SUBAPPLICATION Uebung_036 (* Spiegelabfolge V2 mit Schrittkette *)
  (* Standard: 61499-2; Description: Copyright (c) 2023 Meisterschulen am Ostbahnhof This program and the accompanying materials are made available under the terms of the Eclipse Public License 2.0 which is available at https://www.eclipse.org/legal/epl-2.0/ SPDX-License-Identifier: EPL-2.0 *)
  (* Version 1.0, 2023-10-23, Franz Höpfinger, Meisterschulen am Ostbahnhof *)
  PACKAGE Uebungen;
  IMPORT Uebungen::const::UT::DefaultPool::OutputNumber_N1;
  IMPORT logiBUS::io::DI::logiBUS_DI::Input_I1;
  IMPORT logiBUS::io::DI::logiBUS_DI::Input_I2;
  IMPORT logiBUS::io::DI::logiBUS_DI::Input_I3;
  IMPORT logiBUS::io::DI::logiBUS_DI::Input_I4;
  IMPORT logiBUS::io::DI::logiBUS_DI_Events::BUTTON_SINGLE_CLICK;
  IMPORT logiBUS::io::DQ::logiBUS_DO::Output_Q1;
  IMPORT logiBUS::io::DQ::logiBUS_DO::Output_Q2;
  IMPORT logiBUS::io::DQ::logiBUS_DO::Output_Q3;
  IMPORT logiBUS::io::DQ::logiBUS_DO::Output_Q4;
  IMPORT logiBUS::utils::sequence::const::sequence::NO_TIME;
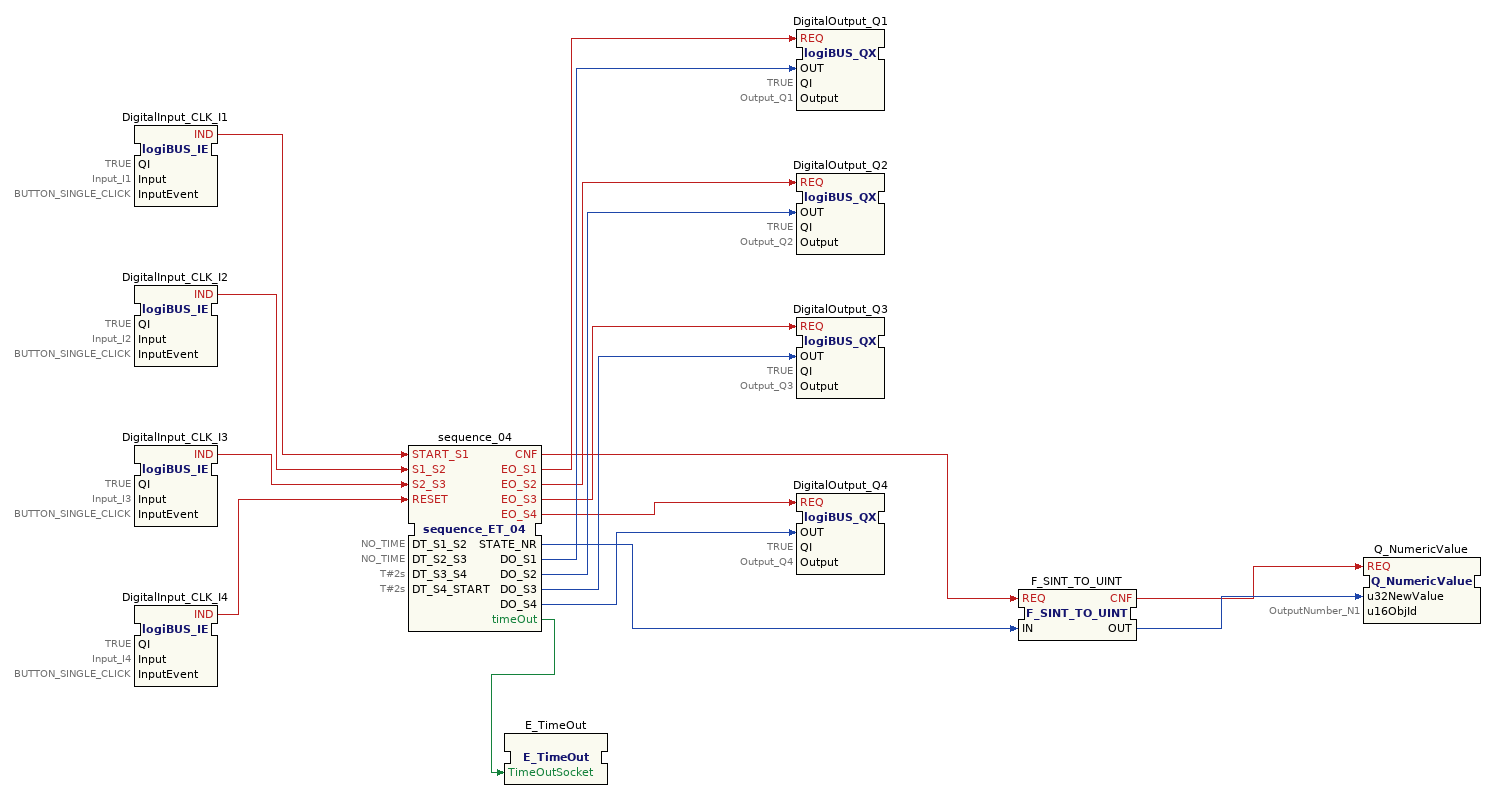
  FBS
    DigitalOutput_Q1 : logiBUS::io::DQ::logiBUS_QX(QI := TRUE, Output := Output_Q1);
    E_TimeOut : iec61499::events::E_TimeOut;
    DigitalOutput_Q2 : logiBUS::io::DQ::logiBUS_QX(QI := TRUE, Output := Output_Q2);
    DigitalOutput_Q3 : logiBUS::io::DQ::logiBUS_QX(QI := TRUE, Output := Output_Q3);
    DigitalOutput_Q4 : logiBUS::io::DQ::logiBUS_QX(QI := TRUE, Output := Output_Q4);
    DigitalInput_CLK_I1 : logiBUS::io::DI::logiBUS_IE(QI := TRUE, Input := Input_I1, InputEvent := BUTTON_SINGLE_CLICK);
    DigitalInput_CLK_I2 : logiBUS::io::DI::logiBUS_IE(QI := TRUE, Input := Input_I2, InputEvent := BUTTON_SINGLE_CLICK);
    DigitalInput_CLK_I3 : logiBUS::io::DI::logiBUS_IE(QI := TRUE, Input := Input_I3, InputEvent := BUTTON_SINGLE_CLICK);
    DigitalInput_CLK_I4 : logiBUS::io::DI::logiBUS_IE(QI := TRUE, Input := Input_I4, InputEvent := BUTTON_SINGLE_CLICK);
    Q_NumericValue : isobus::UT::Q::Q_NumericValue(u16ObjId := OutputNumber_N1);
    F_SINT_TO_UINT : iec61131::conversion::F_SINT_TO_UINT;
    sequence_04 : logiBUS::utils::sequence::combi::sequence_ET_04(DT_S1_S2 := NO_TIME, DT_S2_S3 := NO_TIME, DT_S3_S4 := T#2s, DT_S4_START := T#2s);
  END_FBS
  EVENT_CONNECTIONS
    F_SINT_TO_UINT.CNF TO Q_NumericValue.REQ;
    DigitalInput_CLK_I1.IND TO sequence_04.START_S1;
    DigitalInput_CLK_I2.IND TO sequence_04.S1_S2;
    DigitalInput_CLK_I3.IND TO sequence_04.S2_S3;
    DigitalInput_CLK_I4.IND TO sequence_04.RESET;
    sequence_04.CNF TO F_SINT_TO_UINT.REQ;
    sequence_04.EO_S1 TO DigitalOutput_Q1.REQ;
    sequence_04.EO_S2 TO DigitalOutput_Q2.REQ;
    sequence_04.EO_S3 TO DigitalOutput_Q3.REQ;
    sequence_04.EO_S4 TO DigitalOutput_Q4.REQ;
  END_CONNECTIONS
  DATA_CONNECTIONS
    F_SINT_TO_UINT.OUT TO Q_NumericValue.u32NewValue;
    sequence_04.STATE_NR TO F_SINT_TO_UINT.IN;
    sequence_04.DO_S1 TO DigitalOutput_Q1.OUT;
    sequence_04.DO_S2 TO DigitalOutput_Q2.OUT;
    sequence_04.DO_S3 TO DigitalOutput_Q3.OUT;
    sequence_04.DO_S4 TO DigitalOutput_Q4.OUT;
  END_CONNECTIONS
  ADAPTER_CONNECTIONS
    sequence_04.timeOut TO E_TimeOut.TimeOutSocket;
  END_CONNECTIONS
END_SUBAPPLICATION
